// Mitsubishi GX Works2 project: SVEX   PLC: Q03UDV

PROGRAM MAIN
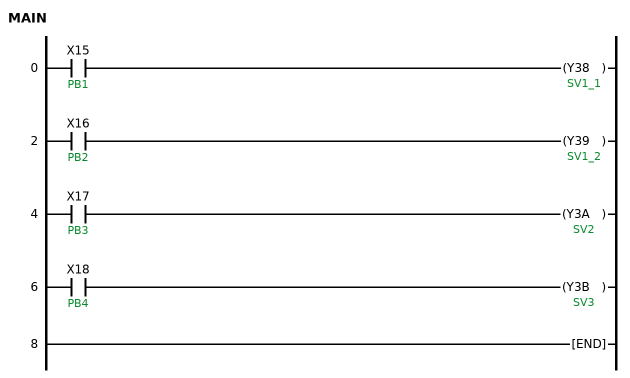
0     LD      X15  ; PB1
      OUT     Y38  ; SV1_1
2     LD      X16  ; PB2
      OUT     Y39  ; SV1_2
4     LD      X17  ; PB3
      OUT     Y3A  ; SV2
6     LD      X18  ; PB4
      OUT     Y3B  ; SV3
8     END
END_PROGRAM

// device comments not shown above
X1  ; PB1
X2  ; PB2
X3  ; PB3
X4  ; PB4
